FUNCTION_BLOCK XCBR_Logic (* Basic Function Block Type *)
  (* Standard: 61499-2 *)
  (* Version 0.0, 12/11/2023, Cheyan, Schneider Electric, Template *)
  PACKAGE Main;
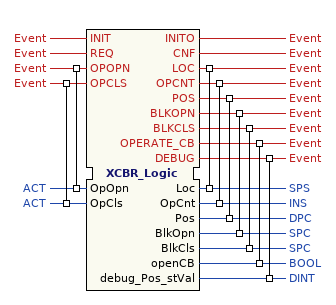
  EVENT_INPUT
    INIT; (* Initialization Request *)
    REQ; (* Normal Execution Request *)
    OPOPN WITH OpOpn;
    OPCLS WITH OpCls;
  END_EVENT
  EVENT_OUTPUT
    INITO; (* Initialization Confirm *)
    CNF; (* Execution Confirmation *)
    LOC WITH Loc;
    OPCNT WITH OpCnt;
    POS WITH Pos;
    BLKOPN WITH BlkOpn;
    BLKCLS WITH BlkCls;
    OPERATE_CB WITH openCB;
    DEBUG WITH debug_Pos_stVal;
  END_EVENT
  VAR_INPUT
    OpOpn : ACT; (* Input event qualifier *)
    OpCls : ACT;
  END_VAR
  VAR_OUTPUT
    Loc : SPS;
    OpCnt : INS;
    Pos : DPC;
    BlkOpn : SPC;
    BlkCls : SPC;
    openCB : BOOL;
    debug_Pos_stVal : DINT;
  END_VAR
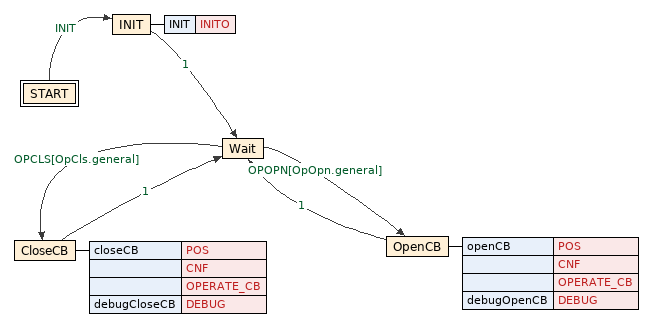
  EC_STATES
    START; (* Initial State *)
    INIT : INIT -> INITO; (* Initialization *)
    Wait; (* Normal execution *)
    OpenCB : openCB -> POS, -> CNF, -> OPERATE_CB, debugOpenCB -> DEBUG;
    CloseCB : closeCB -> POS, -> CNF, -> OPERATE_CB, debugCloseCB -> DEBUG;
  END_STATES
  EC_TRANSITIONS
    START TO INIT := INIT;
    INIT TO Wait := 1;
    Wait TO OpenCB := OPOPN[OpOpn.general];
    OpenCB TO Wait := 1;
    Wait TO CloseCB := OPCLS[OpCls.general];
    CloseCB TO Wait := 1;
  END_TRANSITIONS
  ALGORITHM INIT IN ST: (* Initialization algorithm Setting the initial position of the CB to the "Closed" state stVal is a coded Enum: "1:intermediate-state 2:off 3:on 4:bad-state" *)
;

Pos.stVal := Main.stVal#item3;
  END_ALGORITHM
  ALGORITHM REQ IN ST: (* Normally executed algorithm *)
;
  END_ALGORITHM
  ALGORITHM openCB IN ST: (* To open the CB, set Pos_stVal to false Setting the initial position of the CB to the "opened" state stVal is a coded Enum: "1:intermediate-state 2:off 3:on 4:bad-state" *)
;

Pos.stVal := Main.stVal#item2;

// Open the CB in our plant model
openCB := TRUE;
  END_ALGORITHM
  ALGORITHM closeCB IN ST: (* To close the CB, set Pos_stVal to true Setting the initial position of the CB to the "Closed" state stVal is a coded Enum: "1:intermediate-state 2:off 3:on 4:bad-state" *)
;

Pos.stVal := Main.stVal#item3;

// Close the CB in our plant model
openCB := FALSE;
  END_ALGORITHM
  ALGORITHM debugOpenCB IN ST:
;

debug_Pos_stVal := 2;
  END_ALGORITHM
  ALGORITHM debugCloseCB IN ST:
;

debug_Pos_stVal := 3;
  END_ALGORITHM
END_FUNCTION_BLOCK
